PROGRAM MAIN_SC
VAR
	stTransitions	:	ST_Transitions;
END_VAR

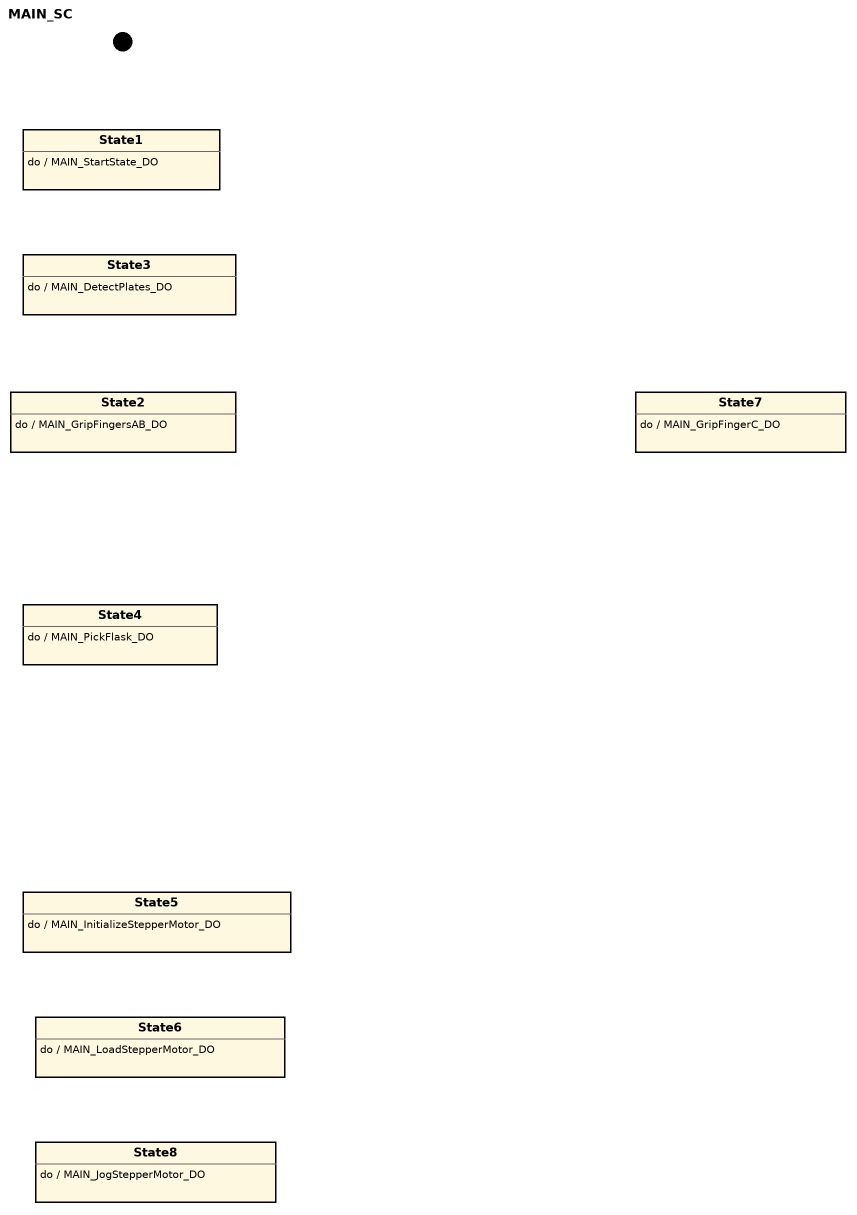
STATECHART MAIN_SC  // abortable
    START StartState1
    STATE State1
        do / MAIN_StartState_DO
    STATE State3
        do / MAIN_DetectPlates_DO
    STATE State2
        do / MAIN_GripFingersAB_DO
    STATE State7
        do / MAIN_GripFingerC_DO
    STATE State4
        do / MAIN_PickFlask_DO
    STATE State5
        do / MAIN_InitializeStepperMotor_DO
    STATE State6
        do / MAIN_LoadStepperMotor_DO
    STATE State8
        do / MAIN_JogStepperMotor_DO
END_STATECHART

ACTION MAIN_DetectPlates_DO:
// Writing Inputs to Robot

// Current Task
END_ACTION

ACTION MAIN_GripFingersAB_DO:

// Resetting Previous state


// Current Task
END_ACTION

ACTION MAIN_GripFingersCD_DO:

// Resetting Previous state


// Current Task
END_ACTION

ACTION MAIN_PickFlask_DO:
// Resetting Previous state
// stTransitions.

// Writing the position of the tablet to the robot registers
// process_gvl.fRobotOutput.General_Register1.Floats.Floats[0] := -0.49657 + (aWorldTabletCoordinates[nTabletCount - 1][0])/1000;
// process_gvl.fRobotOutput.General_Register1.Floats.Floats[1] := 0.04642 + (aWorldTabletCoordinates[nTabletCount - 1][1])/1000;

// Writing Inputs to Robot

// Current Task
// stTransitions.TabletPicked := fbRobot.PickTablet();
END_ACTION

ACTION MAIN_PlaceFlask_DO:

END_ACTION

ACTION MAIN_StartState_DO:
// Read Inputs from Robot

// Write Inputs to Robot

// Reset Values

// Send TaskID to Robot
END_ACTION

END_PROGRAM

(* stored: Version 1.1.0.1
   POU MAIN_SC: Id {2cf27b92-90cd-49d2-a59f-13bef2be8f71}, SpecialFunc None
   Action MAIN_DetectPlates_DO: Id {c2a88684-8b63-4235-8481-da136b8c9166}
   Action MAIN_GripFingersAB_DO: Id {99e88c4b-10e8-43e9-b3a5-8ff6b7c32c58}
   Action MAIN_GripFingersCD_DO: Id {d3c8fdc1-ca0b-48b5-809f-70115616d6e6}
   Action MAIN_PickFlask_DO: Id {210c0cbc-9efe-44c4-bd03-94896909f0d8}
   Action MAIN_PlaceFlask_DO: Id {b2199e2e-eaf7-4c7b-b99e-7656ec0cdd4b}
   Action MAIN_StartState_DO: Id {76120152-bda0-4eed-addf-3629bdd3a69a} *)
